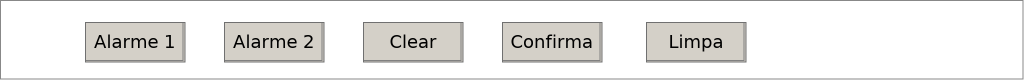
VISUALIZATION Footer  // 1024x80
    Button (85,22 100x40), "Alarme 1"
        toggle prgAlarmHnd.doRaiseEvt1
    Button (224,22 100x40), "Alarme 2"
        toggle prgAlarmHnd.doRaiseEvt2
    Button (363,22 100x40), "Clear"
        tap prgAlarmHnd.doClearEvts
    Button (502,22 100x40), "Confirma"
        tap prgAlarmHnd.doConfirmEvts
    Button (646,22 100x40), "Limpa"
        tap prgAlarmHnd.doClearTable
END_VISUALIZATION

(* stored: Version 1.1.0.1
   Visu Footer: Id {b6e3d4a7-c69e-4564-8ecc-eb462f4bcd95} *)
